VAR_GLOBAL
    //Better have your inputs and outputs!
    // M1L0
    Serial_stComIn_M1L0 AT %I* : EL6inData22B; // M1L0 In Serial Comm Array
    Serial_stComOut_M1L0 AT %Q* : EL6outData22B; // M1L0 Out Serual Comm Array

    // M2L0
    Serial_stComIn_M2L0 AT %I* : EL6inData22B; // M2L0 In Serial Comm Array
    Serial_stComOut_M2L0 AT %Q* : EL6outData22B; // M2L0 Out Serial Comm Array
END_VAR

(* stored: Version 1.1.0.1, ProductVersion 3.1.4022.18
   GVL GVL_SerialIO: Id {e2338c89-1965-407c-b604-590f80e0dc24} *)
